// TIA Portal V19 export
DATA_BLOCK "InstEm2CalledInPreInterpolator"   // DB9
AUTHOR : Siemens_FA_SUP
// stored: InstanceOfName Unit.Em2.CalledInPreInterpolator, InstanceOfType FB
"Unit.Em2.CalledInPreInterpolator"
BEGIN
END_DATA_BLOCK
